(* IEC 61131-3 sources: RL_MAR/experiments/comparison/llm4plc/results/gpt-4o-mini_20260506_100619/20260506_102515, 4 files *)

(* ---- generated_code_iteration_0.st ---- *)
ructured-text
FUNCTION_BLOCK CarParkingSystem
VAR_INPUT
    NewCarSlot : INT; (* Input for new car arrival slot number *)
END_VAR
VAR_OUTPUT
    Elevator1Busy : BOOL; (* Elevator 1 status - busy or idle *)
    Elevator2Busy : BOOL; (* Elevator 2 status - busy or idle *)
    Elevator1Position : INT; (* Elevator 1 current position *)
    Elevator2Position : INT; (* Elevator 2 current position *)
END_VAR
VAR
    Elevator1Target : INT; (* Elevator 1 target floor *)
    Elevator2Target : INT; (* Elevator 2 target floor *)
    CarSlots : ARRAY[1..100] OF BOOL; (* Array to represent parking slots - TRUE if occupied *)
    CurrentSlot : INT; (* Loop counter for scanning slots *)
    state : INT; (* The state variable *)
    prevState : INT; (* The previous state variable *)
END_VAR

(* State Definitions *)
CONST
    IDLE : INT := 0;
    ASSIGN_ELEVATOR : INT := 1;
    MOVE_ELEVATOR : INT := 2;
    PARK_CAR : INT := 3;
    SCAN_SLOTS : INT := 4;
END_CONST

(* Initialization *)
state := IDLE;
prevState := IDLE;

(* State Machine Implementation *)
CASE state OF
    IDLE:
        Elevator1Busy := FALSE;
        Elevator2Busy := FALSE;
        Elevator1Position := Elevator1Position; (* Current position remains unchanged *)
        Elevator2Position := Elevator2Position; (* Current position remains unchanged *)

        IF NewCarSlot <> 0 THEN
            state := SCAN_SLOTS; (* Transition to scanning slots for new car *)
        END_IF

    SCAN_SLOTS:
        IF NOT CarSlots[NewCarSlot] THEN
            state := ASSIGN_ELEVATOR; (* Transition to assign elevator if slot is free *)
        ELSE
            state := IDLE; (* Stay in IDLE if slot is occupied *)
        END_IF

    ASSIGN_ELEVATOR:
        IF NewCarSlot <= 50 THEN
            Elevator1Target := NewCarSlot; (* Assign Elevator 1 for slots 1-50 *)
            Elevator1Busy := TRUE;
        ELSE
            Elevator2Target := NewCarSlot; (* Assign Elevator 2 for slots 51-100 *)
            Elevator2Busy := TRUE;
        END_IF

        IF Elevator1Busy OR Elevator2Busy THEN
            state := MOVE_ELEVATOR; (* Transition to move elevator if assigned *)
        END_IF

    MOVE_ELEVATOR:
        IF (Elevator1Busy AND Elevator1Position = Elevator1Target) OR
           (Elevator2Busy AND Elevator2Position = Elevator2Target) THEN
            state := PARK_CAR; (* Transition to park car if elevator reached target *)
        END_IF

    PARK_CAR:
        CarSlots[NewCarSlot] := TRUE; (* Mark the parking slot as occupied *)
        IF Elevator1Busy THEN
            Elevator1Busy := FALSE; (* Elevator 1 is now idle after parking *)
        END_IF
        IF Elevator2Busy THEN
            Elevator2Busy := FALSE; (* Elevator 2 is now idle after parking *)
        END_IF
        state := IDLE; (* Return to IDLE state after parking the car *)

END_CASE

END_FUNCTION_BLOCK

(* ---- generated_code_iteration_1.st ---- *)
START_REASON
The errors occurred due to the incorrect use of a colon (:) instead of a semicolon (;) in the state machine implementation. Specifically, the line where the state variable is assigned the value of IDLE should use a semicolon to terminate the statement. This is a syntax requirement in Structured Text (ST) programming.
END_REASON

START_ST
FUNCTION_BLOCK CarParkingSystem
VAR_INPUT
    NewCarSlot : INT; (* Input for new car arrival slot number *)
END_VAR
VAR_OUTPUT
    Elevator1Busy : BOOL; (* Elevator 1 status - busy or idle *)
    Elevator2Busy : BOOL; (* Elevator 2 status - busy or idle *)
    Elevator1Position : INT; (* Elevator 1 current position *)
    Elevator2Position : INT; (* Elevator 2 current position *)
END_VAR
VAR
    Elevator1Target : INT; (* Elevator 1 target floor *)
    Elevator2Target : INT; (* Elevator 2 target floor *)
    CarSlots : ARRAY[1..100] OF BOOL; (* Array to represent parking slots - TRUE if occupied *)
    CurrentSlot : INT; (* Loop counter for scanning slots *)
    state : INT; (* The state variable *)
    prevState : INT; (* The previous state variable *)
END_VAR

(* State Definitions *)
CONST
    IDLE : INT := 0;
    ASSIGN_ELEVATOR : INT := 1;
    MOVE_ELEVATOR : INT := 2;
    PARK_CAR : INT := 3;
    SCAN_SLOTS : INT := 4;
END_CONST

(* Initialization *)
state := IDLE;
prevState := IDLE;

(* State Machine Implementation *)
CASE state OF
    IDLE:
        Elevator1Busy := FALSE;
        Elevator2Busy := FALSE;
        Elevator1Position := Elevator1Position; (* Current position remains unchanged *)
        Elevator2Position := Elevator2Position; (* Current position remains unchanged *)

        IF NewCarSlot <> 0 THEN
            state := SCAN_SLOTS; (* Transition to scanning slots for new car *)
        END_IF;

    SCAN_SLOTS:
        IF NOT CarSlots[NewCarSlot] THEN
            state := ASSIGN_ELEVATOR; (* Transition to assign elevator if slot is free *)
        ELSE
            state := IDLE; (* Stay in IDLE if slot is occupied *)
        END_IF;

    ASSIGN_ELEVATOR:
        IF NewCarSlot <= 50 THEN
            Elevator1Target := NewCarSlot; (* Assign Elevator 1 for slots 1-50 *)
            Elevator1Busy := TRUE;
        ELSE
            Elevator2Target := NewCarSlot; (* Assign Elevator 2 for slots 51-100 *)
            Elevator2Busy := TRUE;
        END_IF;

        IF Elevator1Busy OR Elevator2Busy THEN
            state := MOVE_ELEVATOR; (* Transition to move elevator if assigned *)
        END_IF;

    MOVE_ELEVATOR:
        IF (Elevator1Busy AND Elevator1Position = Elevator1Target) OR
           (Elevator2Busy AND Elevator2Position = Elevator2Target) THEN
            state := PARK_CAR; (* Transition to park car if elevator reached target *)
        END_IF;

    PARK_CAR:
        CarSlots[NewCarSlot] := TRUE; (* Mark the parking slot as occupied *)
        IF Elevator1Busy THEN
            Elevator1Busy := FALSE; (* Elevator 1 is now idle after parking *)
        END_IF;
        IF Elevator2Busy THEN
            Elevator2Busy := FALSE; (* Elevator 2 is now idle after parking *)
        END_IF;
        state := IDLE; (* Return to IDLE state after parking the car *)

END_CASE;

END_FUNCTION_BLOCK
END_ST

(* ---- generated_code_iteration_2.st ---- *)
START_REASON
The errors occurred due to the incorrect use of a colon (:) instead of a semicolon (;) in the state machine implementation. Specifically, the line where the state variable is assigned the value of IDLE should use a semicolon to terminate the statement. This is a syntax requirement in Structured Text (ST) programming.
END_REASON

START_ST
FUNCTION_BLOCK CarParkingSystem
VAR_INPUT
    NewCarSlot : INT; (* Input for new car arrival slot number *)
END_VAR
VAR_OUTPUT
    Elevator1Busy : BOOL; (* Elevator 1 status - busy or idle *)
    Elevator2Busy : BOOL; (* Elevator 2 status - busy or idle *)
    Elevator1Position : INT; (* Elevator 1 current position *)
    Elevator2Position : INT; (* Elevator 2 current position *)
END_VAR
VAR
    Elevator1Target : INT; (* Elevator 1 target floor *)
    Elevator2Target : INT; (* Elevator 2 target floor *)
    CarSlots : ARRAY[1..100] OF BOOL; (* Array to represent parking slots - TRUE if occupied *)
    CurrentSlot : INT; (* Loop counter for scanning slots *)
    state : INT; (* The state variable *)
    prevState : INT; (* The previous state variable *)
END_VAR

(* State Definitions *)
CONST
    IDLE : INT := 0;
    ASSIGN_ELEVATOR : INT := 1;
    MOVE_ELEVATOR : INT := 2;
    PARK_CAR : INT := 3;
    SCAN_SLOTS : INT := 4;
END_CONST

(* Initialization *)
state := IDLE;
prevState := IDLE;

(* State Machine Implementation *)
CASE state OF
    IDLE:
        Elevator1Busy := FALSE;
        Elevator2Busy := FALSE;
        Elevator1Position := Elevator1Position; (* Current position remains unchanged *)
        Elevator2Position := Elevator2Position; (* Current position remains unchanged *)

        IF NewCarSlot <> 0 THEN
            state := SCAN_SLOTS; (* Transition to scanning slots for new car *)
        END_IF;

    SCAN_SLOTS:
        IF NOT CarSlots[NewCarSlot] THEN
            state := ASSIGN_ELEVATOR; (* Transition to assign elevator if slot is free *)
        ELSE
            state := IDLE; (* Stay in IDLE if slot is occupied *)
        END_IF;

    ASSIGN_ELEVATOR:
        IF NewCarSlot <= 50 THEN
            Elevator1Target := NewCarSlot; (* Assign Elevator 1 for slots 1-50 *)
            Elevator1Busy := TRUE;
        ELSE
            Elevator2Target := NewCarSlot; (* Assign Elevator 2 for slots 51-100 *)
            Elevator2Busy := TRUE;
        END_IF;

        IF Elevator1Busy OR Elevator2Busy THEN
            state := MOVE_ELEVATOR; (* Transition to move elevator if assigned *)
        END_IF;

    MOVE_ELEVATOR:
        IF (Elevator1Busy AND Elevator1Position = Elevator1Target) OR
           (Elevator2Busy AND Elevator2Position = Elevator2Target) THEN
            state := PARK_CAR; (* Transition to park car if elevator reached target *)
        END_IF;

    PARK_CAR:
        CarSlots[NewCarSlot] := TRUE; (* Mark the parking slot as occupied *)
        IF Elevator1Busy THEN
            Elevator1Busy := FALSE; (* Elevator 1 is now idle after parking *)
        END_IF;
        IF Elevator2Busy THEN
            Elevator2Busy := FALSE; (* Elevator 2 is now idle after parking *)
        END_IF;
        state := IDLE; (* Return to IDLE state after parking the car *)

END_CASE;

END_FUNCTION_BLOCK
END_ST

(* ---- generated_code_iteration_3.st ---- *)
START_REASON
The errors occurred due to the incorrect use of a colon (:) instead of a semicolon (;) in the state machine implementation. Specifically, the line where the state variable is assigned the value of IDLE should use a semicolon to terminate the statement. This is a syntax requirement in Structured Text (ST) programming. The code also needs to ensure that all statements are properly terminated with semicolons to comply with ST syntax rules.
END_REASON

START_ST
FUNCTION_BLOCK CarParkingSystem
VAR_INPUT
    NewCarSlot : INT; (* Input for new car arrival slot number *)
END_VAR
VAR_OUTPUT
    Elevator1Busy : BOOL; (* Elevator 1 status - busy or idle *)
    Elevator2Busy : BOOL; (* Elevator 2 status - busy or idle *)
    Elevator1Position : INT; (* Elevator 1 current position *)
    Elevator2Position : INT; (* Elevator 2 current position *)
END_VAR
VAR
    Elevator1Target : INT; (* Elevator 1 target floor *)
    Elevator2Target : INT; (* Elevator 2 target floor *)
    CarSlots : ARRAY[1..100] OF BOOL; (* Array to represent parking slots - TRUE if occupied *)
    CurrentSlot : INT; (* Loop counter for scanning slots *)
    state : INT; (* The state variable *)
    prevState : INT; (* The previous state variable *)
END_VAR

(* State Definitions *)
CONST
    IDLE : INT := 0;
    ASSIGN_ELEVATOR : INT := 1;
    MOVE_ELEVATOR : INT := 2;
    PARK_CAR : INT := 3;
    SCAN_SLOTS : INT := 4;
END_CONST

(* Initialization *)
state := IDLE; (* Corrected with semicolon *)
prevState := IDLE; (* Corrected with semicolon *)

(* State Machine Implementation *)
CASE state OF
    IDLE:
        Elevator1Busy := FALSE;
        Elevator2Busy := FALSE;
        Elevator1Position := Elevator1Position; (* Current position remains unchanged *)
        Elevator2Position := Elevator2Position; (* Current position remains unchanged *)

        IF NewCarSlot <> 0 THEN
            state := SCAN_SLOTS; (* Transition to scanning slots for new car *)
        END_IF;

    SCAN_SLOTS:
        IF NOT CarSlots[NewCarSlot] THEN
            state := ASSIGN_ELEVATOR; (* Transition to assign elevator if slot is free *)
        ELSE
            state := IDLE; (* Stay in IDLE if slot is occupied *)
        END_IF;

    ASSIGN_ELEVATOR:
        IF NewCarSlot <= 50 THEN
            Elevator1Target := NewCarSlot; (* Assign Elevator 1 for slots 1-50 *)
            Elevator1Busy := TRUE;
        ELSE
            Elevator2Target := NewCarSlot; (* Assign Elevator 2 for slots 51-100 *)
            Elevator2Busy := TRUE;
        END_IF;

        IF Elevator1Busy OR Elevator2Busy THEN
            state := MOVE_ELEVATOR; (* Transition to move elevator if assigned *)
        END_IF;

    MOVE_ELEVATOR:
        IF (Elevator1Busy AND Elevator1Position = Elevator1Target) OR
           (Elevator2Busy AND Elevator2Position = Elevator2Target) THEN
            state := PARK_CAR; (* Transition to park car if elevator reached target *)
        END_IF;

    PARK_CAR:
        CarSlots[NewCarSlot] := TRUE; (* Mark the parking slot as occupied *)
        IF Elevator1Busy THEN
            Elevator1Busy := FALSE; (* Elevator 1 is now idle after parking *)
        END_IF;
        IF Elevator2Busy THEN
            Elevator2Busy := FALSE; (* Elevator 2 is now idle after parking *)
        END_IF;
        state := IDLE; (* Return to IDLE state after parking the car *)

END_CASE;

END_FUNCTION_BLOCK
END_ST
